{attribute 'linkalways'} 
{attribute 'no_explicit_call' := 'This FB is a CLASS and must be accessed using methods or properties'}
{attribute 'enable_dynamic_creation'}
FUNCTION_BLOCK Node_F_VN_ExportImageAsBmpSize EXTENDS VisionNode
VAR
    ipImage : _ITcVnImage;
    nBufferSize : _ULINT(0);
    hrPrev : _HRESULT(S_OK);
	hresult : _HRESULT(S_OK);
END_VAR

METHOD PUBLIC  Clone : I_Node
VAR
	pNode : POINTER TO Node_F_VN_ExportImageAsBmpSize;
END_VAR
pNode := __NEW(Node_F_VN_ExportImageAsBmpSize);
Clone := pNode^;
END_METHOD

METHOD FB_init : BOOL
VAR_INPUT
	bInitRetains : BOOL; // if TRUE, the retain variables are initialized (warm start / cold start)
	bInCopyCode : BOOL;  // if TRUE, the instance afterwards gets moved into the copy code (online change)
END_VAR
AddInput('ipImage', ipImage);
AddInput('hrPrev', hrPrev);
AddOutput('nBufferSize', nBufferSize);
AddOutput('hresult',hresult);
END_METHOD

METHOD PROTECTED  OnExecute : HRESULT
hresult.Value := F_VN_ExportImageAsBmpSize(
    ipImage := ipImage.Value,
    nBufferSize := nBufferSize.Value,
	hrPrev:= hrPrev.Value);
END_METHOD

METHOD PUBLIC PreExecutionCheck
VAR_INPUT
	Check : I_PreExecutionChecks;
END_VAR
Check.IsTrue(ipImage.IsValid, 'ipImage must contain an image');
END_METHOD

END_FUNCTION_BLOCK

(* stored: Version 1.1.0.1, ProductVersion 3.1.4024.13
   POU Node_F_VN_ExportImageAsBmpSize: Id {9746f255-7be7-0b43-23b2-77277bbff7ea}, SpecialFunc None
   Folder Constructor: Id {fe01235c-ecb5-02e8-212c-68b370171c71}
   Method Clone: Id {86556fbe-fc8b-0895-3bfd-abbf29fd4390}
   Method FB_init: Id {9e190ed5-662e-07c0-3cd6-539fd1260518}
   Method OnExecute: Id {43851544-f7b5-0156-0a73-0ac6f15c5639}
   Method PreExecutionCheck: Id {c12afd70-ac43-03c9-0e9f-57fee57689b7} *)
